FUNCTION_BLOCK F_SEL_E_2 (* selection (event-based selection) *)
  (* Standard: 61131-3; Classification: standard selection function; Description: Copyright (c) 2012, 2022 TU Wien ACIN, HR Agrartechnik GmbH This program and the accompanying materials are made available under the terms of the Eclipse Public License 2.0 which is available at https://www.eclipse.org/legal/epl-2.0/ SPDX-License-Identifier: EPL-2.0 *)
  (* Version 1.0, 2012-03-25, Monika Wenger, TU Wien ACIN *)
  (* Version 1.1, 2022-08-04, Franz Höpfinger, HR Agrartechnik GmbH *)
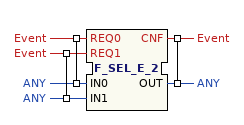
  EVENT_INPUT
    REQ0 WITH IN0;
    REQ1 WITH IN1;
  END_EVENT
  EVENT_OUTPUT
    CNF WITH OUT; (* Confirmation of Requested Service *)
  END_EVENT
  VAR_INPUT
    IN0 : ANY; (* Selectable input variable *)
    IN1 : ANY; (* Selectable input variable *)
  END_VAR
  VAR_OUTPUT
    OUT : ANY; (* Selected input *)
  END_VAR
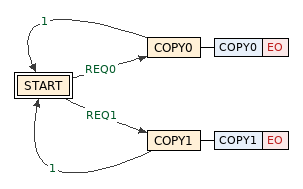
  EC_STATES
    START; (* Initial State *)
    COPY0 : COPY0 -> EO;
    COPY1 : COPY1 -> EO;
  END_STATES
  EC_TRANSITIONS
    START TO COPY0 := REQ0;
    START TO COPY1 := REQ1;
    COPY0 TO START := 1;
    COPY1 TO START := 1;
  END_TRANSITIONS
  ALGORITHM COPY0 IN ST:
OUT := IN0;
  END_ALGORITHM
  ALGORITHM COPY1 IN ST:
OUT := IN1;
  END_ALGORITHM
END_FUNCTION_BLOCK
